Staubli VAL3: getY.pgx

public program getY(num& nValueY (dimensions=1))
  local point pHere
begin
  pHere=here(tActive,frActive)
  nValueY=pHere.trsf.y
end
